(* IEC 61131-3 sources: ST2CPP/java/src/main/resources, 1 file *)

(* ---- iec_stdlib.st ---- *)
(* IEC 61131-3 标准类型转换函数声明 *)
(* 编译器生成 C++ 原型，运行时在 rt_plc.h 中实现 *)
(* 注意: TIME_OF_DAY/DATE_AND_TIME 类型暂不被 parser 识别，用 DINT/STRING 替代 *)

(* ─── 类型转换: X_TO_Y ─── *)
FUNCTION DINT_TO_TIME : TIME VAR_INPUT IN : DINT; END_VAR END_FUNCTION
FUNCTION UDINT_TO_DINT : DINT VAR_INPUT IN : UDINT; END_VAR END_FUNCTION
FUNCTION INT_TO_UDINT : UDINT VAR_INPUT IN : INT; END_VAR END_FUNCTION
FUNCTION UDINT_TO_TIME : TIME VAR_INPUT IN : UDINT; END_VAR END_FUNCTION
FUNCTION DINT_TO_UDINT : UDINT VAR_INPUT IN : DINT; END_VAR END_FUNCTION
FUNCTION TIME_TO_UDINT : UDINT VAR_INPUT IN : TIME; END_VAR END_FUNCTION
FUNCTION REAL_TO_DINT : DINT VAR_INPUT IN : REAL; END_VAR END_FUNCTION
FUNCTION REAL_TO_UDINT : UDINT VAR_INPUT IN : REAL; END_VAR END_FUNCTION
FUNCTION REAL_TO_DWORD : DWORD VAR_INPUT IN : REAL; END_VAR END_FUNCTION
FUNCTION REAL_TO_INT : INT VAR_INPUT IN : REAL; END_VAR END_FUNCTION
FUNCTION REAL_TO_WORD : WORD VAR_INPUT IN : REAL; END_VAR END_FUNCTION
FUNCTION REAL_TO_BYTE : BYTE VAR_INPUT IN : REAL; END_VAR END_FUNCTION
FUNCTION REAL_TO_TIME : TIME VAR_INPUT IN : REAL; END_VAR END_FUNCTION
FUNCTION REAL_TO_STRF : STRING VAR_INPUT IN : REAL; END_VAR END_FUNCTION
FUNCTION REAL_TO_STRING : STRING VAR_INPUT IN : REAL; END_VAR END_FUNCTION
FUNCTION INT_TO_DINT : DINT VAR_INPUT IN : INT; END_VAR END_FUNCTION
FUNCTION INT_TO_REAL : REAL VAR_INPUT IN : INT; END_VAR END_FUNCTION
FUNCTION INT_TO_DWORD : DWORD VAR_INPUT IN : INT; END_VAR END_FUNCTION
FUNCTION INT_TO_BYTE : BYTE VAR_INPUT IN : INT; END_VAR END_FUNCTION
FUNCTION INT_TO_WORD : WORD VAR_INPUT IN : INT; END_VAR END_FUNCTION
FUNCTION INT_TO_STRING : STRING VAR_INPUT IN : INT; END_VAR END_FUNCTION
FUNCTION INT_TO_TIME : TIME VAR_INPUT IN : INT; END_VAR END_FUNCTION
FUNCTION INT_TO_UINT : UINT VAR_INPUT IN : INT; END_VAR END_FUNCTION
FUNCTION DINT_TO_INT : INT VAR_INPUT IN : DINT; END_VAR END_FUNCTION
FUNCTION DINT_TO_REAL : REAL VAR_INPUT IN : DINT; END_VAR END_FUNCTION
FUNCTION DINT_TO_DWORD : DWORD VAR_INPUT IN : DINT; END_VAR END_FUNCTION
FUNCTION DINT_TO_WORD : WORD VAR_INPUT IN : DINT; END_VAR END_FUNCTION
FUNCTION DINT_TO_STRING : STRING VAR_INPUT IN : DINT; END_VAR END_FUNCTION
FUNCTION DWORD_TO_DINT : DINT VAR_INPUT IN : DWORD; END_VAR END_FUNCTION
FUNCTION DWORD_TO_INT : INT VAR_INPUT IN : DWORD; END_VAR END_FUNCTION
FUNCTION DWORD_TO_WORD : WORD VAR_INPUT IN : DWORD; END_VAR END_FUNCTION
FUNCTION DWORD_TO_BYTE : BYTE VAR_INPUT IN : DWORD; END_VAR END_FUNCTION
FUNCTION DWORD_TO_TIME : TIME VAR_INPUT IN : DWORD; END_VAR END_FUNCTION
FUNCTION DWORD_TO_UDINT : UDINT VAR_INPUT IN : DWORD; END_VAR END_FUNCTION
FUNCTION DWORD_TO_STRING : STRING VAR_INPUT IN : DWORD; END_VAR END_FUNCTION
FUNCTION DWORD_TO_STRB : STRING VAR_INPUT IN : DWORD; END_VAR END_FUNCTION
FUNCTION DWORD_TO_STRH : STRING VAR_INPUT IN : DWORD; END_VAR END_FUNCTION
FUNCTION DWORD_TO_STRF : STRING VAR_INPUT IN : DWORD; END_VAR END_FUNCTION
FUNCTION DW_TO_REAL : REAL VAR_INPUT IN : DWORD; END_VAR END_FUNCTION
FUNCTION UDINT_TO_REAL : REAL VAR_INPUT IN : UDINT; END_VAR END_FUNCTION
FUNCTION UDINT_TO_INT : INT VAR_INPUT IN : UDINT; END_VAR END_FUNCTION
FUNCTION UDINT_TO_DWORD : DWORD VAR_INPUT IN : UDINT; END_VAR END_FUNCTION
FUNCTION UDINT_TO_WORD : WORD VAR_INPUT IN : UDINT; END_VAR END_FUNCTION
FUNCTION UDINT_TO_BYTE : BYTE VAR_INPUT IN : UDINT; END_VAR END_FUNCTION
FUNCTION UDINT_TO_STRING : STRING VAR_INPUT IN : UDINT; END_VAR END_FUNCTION
FUNCTION UDINT_TO_UINT : UINT VAR_INPUT IN : UDINT; END_VAR END_FUNCTION
FUNCTION WORD_TO_DINT : DINT VAR_INPUT IN : WORD; END_VAR END_FUNCTION
FUNCTION WORD_TO_INT : INT VAR_INPUT IN : WORD; END_VAR END_FUNCTION
FUNCTION WORD_TO_DWORD : DWORD VAR_INPUT IN : WORD; END_VAR END_FUNCTION
FUNCTION WORD_TO_BYTE : BYTE VAR_INPUT IN : WORD; END_VAR END_FUNCTION
FUNCTION WORD_TO_UDINT : UDINT VAR_INPUT IN : WORD; END_VAR END_FUNCTION
FUNCTION WORD_TO_UINT : UINT VAR_INPUT IN : WORD; END_VAR END_FUNCTION
FUNCTION WORD_TO_STRING : STRING VAR_INPUT IN : WORD; END_VAR END_FUNCTION
FUNCTION BYTE_TO_DINT : DINT VAR_INPUT IN : BYTE; END_VAR END_FUNCTION
FUNCTION BYTE_TO_INT : INT VAR_INPUT IN : BYTE; END_VAR END_FUNCTION
FUNCTION BYTE_TO_DWORD : DWORD VAR_INPUT IN : BYTE; END_VAR END_FUNCTION
FUNCTION BYTE_TO_WORD : WORD VAR_INPUT IN : BYTE; END_VAR END_FUNCTION
FUNCTION BYTE_TO_UDINT : UDINT VAR_INPUT IN : BYTE; END_VAR END_FUNCTION
FUNCTION BYTE_TO_UINT : UINT VAR_INPUT IN : BYTE; END_VAR END_FUNCTION
FUNCTION BYTE_TO_USINT : USINT VAR_INPUT IN : BYTE; END_VAR END_FUNCTION
FUNCTION BYTE_TO_STRING : STRING VAR_INPUT IN : BYTE; END_VAR END_FUNCTION
FUNCTION BYTE_TO_STRB : STRING VAR_INPUT IN : BYTE; END_VAR END_FUNCTION
FUNCTION BYTE_TO_STRH : STRING VAR_INPUT IN : BYTE; END_VAR END_FUNCTION
FUNCTION BYTE_TO_BITS : STRING VAR_INPUT IN : BYTE; END_VAR END_FUNCTION
FUNCTION BYTE_TO_GRAY : BYTE VAR_INPUT IN : BYTE; END_VAR END_FUNCTION
FUNCTION BYTE_TO_TIME2 : TIME VAR_INPUT IN : BYTE; END_VAR END_FUNCTION
FUNCTION UINT_TO_DINT : DINT VAR_INPUT IN : UINT; END_VAR END_FUNCTION
FUNCTION UINT_TO_INT : INT VAR_INPUT IN : UINT; END_VAR END_FUNCTION
FUNCTION UINT_TO_DWORD : DWORD VAR_INPUT IN : UINT; END_VAR END_FUNCTION
FUNCTION UINT_TO_BYTE : BYTE VAR_INPUT IN : UINT; END_VAR END_FUNCTION
FUNCTION UINT_TO_WORD : WORD VAR_INPUT IN : UINT; END_VAR END_FUNCTION
FUNCTION UINT_TO_UDINT : UDINT VAR_INPUT IN : UINT; END_VAR END_FUNCTION
FUNCTION UINT_TO_REAL : REAL VAR_INPUT IN : UINT; END_VAR END_FUNCTION
FUNCTION USINT_TO_INT : INT VAR_INPUT IN : USINT; END_VAR END_FUNCTION
FUNCTION USINT_TO_BYTE : BYTE VAR_INPUT IN : USINT; END_VAR END_FUNCTION
FUNCTION USINT_TO_REAL : REAL VAR_INPUT IN : USINT; END_VAR END_FUNCTION
FUNCTION USINT_TO_DINT : DINT VAR_INPUT IN : USINT; END_VAR END_FUNCTION
FUNCTION SINT_TO_INT : INT VAR_INPUT IN : SINT; END_VAR END_FUNCTION
FUNCTION SINT_TO_DINT : DINT VAR_INPUT IN : SINT; END_VAR END_FUNCTION
FUNCTION STRING_TO_TIME : TIME VAR_INPUT IN : STRING; END_VAR END_FUNCTION
FUNCTION STRING_TO_INT : INT VAR_INPUT IN : STRING; END_VAR END_FUNCTION
FUNCTION STRING_TO_REAL : REAL VAR_INPUT IN : STRING; END_VAR END_FUNCTION
FUNCTION STRING_TO_DWORD : DWORD VAR_INPUT IN : STRING; END_VAR END_FUNCTION
FUNCTION STRING_TO_WORD : WORD VAR_INPUT IN : STRING; END_VAR END_FUNCTION
FUNCTION STRING_TO_UDINT : UDINT VAR_INPUT IN : STRING; END_VAR END_FUNCTION
FUNCTION STRING_TO_URL : STRING VAR_INPUT IN : STRING; END_VAR END_FUNCTION
FUNCTION STRING_TO_BUFFER : STRING VAR_INPUT IN : STRING; END_VAR END_FUNCTION
FUNCTION BOOL_TO_BYTE : BYTE VAR_INPUT IN : BOOL; END_VAR END_FUNCTION
FUNCTION BOOL_TO_INT : INT VAR_INPUT IN : BOOL; END_VAR END_FUNCTION
FUNCTION BOOL_TO_DWORD : DWORD VAR_INPUT IN : BOOL; END_VAR END_FUNCTION
FUNCTION BOOL_TO_UDINT : UDINT VAR_INPUT IN : BOOL; END_VAR END_FUNCTION
FUNCTION BOOL_TO_STRING : STRING VAR_INPUT IN : BOOL; END_VAR END_FUNCTION
FUNCTION TIME_TO_DINT : DINT VAR_INPUT IN : TIME; END_VAR END_FUNCTION
FUNCTION TIME_TO_INT : INT VAR_INPUT IN : TIME; END_VAR END_FUNCTION
FUNCTION TIME_TO_DWORD : DWORD VAR_INPUT IN : TIME; END_VAR END_FUNCTION
FUNCTION TIME_TO_REAL : REAL VAR_INPUT IN : TIME; END_VAR END_FUNCTION
FUNCTION TIME_TO_TOD : STRING VAR_INPUT IN : TIME; END_VAR END_FUNCTION
FUNCTION TOD_TO_TIME : TIME VAR_INPUT IN : STRING; END_VAR END_FUNCTION
FUNCTION TOD_TO_REAL2 : REAL VAR_INPUT IN : STRING; END_VAR END_FUNCTION
FUNCTION DATE_TO_UDINT : UDINT VAR_INPUT IN : INT; END_VAR END_FUNCTION
FUNCTION DATE_TO_DT : INT VAR_INPUT IN : INT; END_VAR END_FUNCTION
FUNCTION DATE_TO_STRING2 : STRING VAR_INPUT IN : INT; END_VAR END_FUNCTION
FUNCTION DATE_TO_REAL2 : REAL VAR_INPUT IN : INT; END_VAR END_FUNCTION
FUNCTION DATE_TO_DWORD2 : DWORD VAR_INPUT IN : INT; END_VAR END_FUNCTION
FUNCTION DT_TO_DATE : INT VAR_INPUT IN : INT; END_VAR END_FUNCTION
FUNCTION DT_TO_DATE2 : INT VAR_INPUT IN : INT; END_VAR END_FUNCTION
FUNCTION DT_TO_TOD2 : STRING VAR_INPUT IN : INT; END_VAR END_FUNCTION
FUNCTION DT_TO_SDT : INT VAR_INPUT IN : INT; END_VAR END_FUNCTION
FUNCTION DT_TO_STRF : STRING VAR_INPUT IN : INT; END_VAR END_FUNCTION
FUNCTION SDT_TO_DATE : INT VAR_INPUT IN : INT; END_VAR END_FUNCTION
FUNCTION SDT_TO_DT : INT VAR_INPUT IN : INT; END_VAR END_FUNCTION
FUNCTION SDT_TO_TOD : STRING VAR_INPUT IN : INT; END_VAR END_FUNCTION

(* ─── 字符串操作 ─── *)
FUNCTION CONCAT : STRING VAR_INPUT A : STRING; B : STRING; END_VAR END_FUNCTION
FUNCTION LEN : DINT VAR_INPUT S : STRING; END_VAR END_FUNCTION
FUNCTION LEFT : STRING VAR_INPUT S : STRING; L : DINT; END_VAR END_FUNCTION
FUNCTION RIGHT : STRING VAR_INPUT S : STRING; L : DINT; END_VAR END_FUNCTION
FUNCTION MID : STRING VAR_INPUT S : STRING; L : DINT; P : DINT; END_VAR END_FUNCTION
FUNCTION INSERT : STRING VAR_INPUT S : STRING; INS : STRING; P : DINT; END_VAR END_FUNCTION
FUNCTION DELETE : STRING VAR_INPUT S : STRING; L : DINT; P : DINT; END_VAR END_FUNCTION
FUNCTION REPLACE : STRING VAR_INPUT S : STRING; L : DINT; P : DINT; R : STRING; END_VAR END_FUNCTION
FUNCTION FIND : DINT VAR_INPUT S : STRING; SUBSTR : STRING; END_VAR END_FUNCTION
FUNCTION STR_EQ : BOOL VAR_INPUT A : STRING; B : STRING; END_VAR END_FUNCTION
FUNCTION STR_NE : BOOL VAR_INPUT A : STRING; B : STRING; END_VAR END_FUNCTION
FUNCTION STR_LT : BOOL VAR_INPUT A : STRING; B : STRING; END_VAR END_FUNCTION
FUNCTION STR_LE : BOOL VAR_INPUT A : STRING; B : STRING; END_VAR END_FUNCTION
FUNCTION STR_GT : BOOL VAR_INPUT A : STRING; B : STRING; END_VAR END_FUNCTION
FUNCTION STR_GE : BOOL VAR_INPUT A : STRING; B : STRING; END_VAR END_FUNCTION

(* ─── 数学函数 ─── *)
FUNCTION ABS : REAL VAR_INPUT X : REAL; END_VAR END_FUNCTION
FUNCTION SQRT : REAL VAR_INPUT X : REAL; END_VAR END_FUNCTION
FUNCTION LN : REAL VAR_INPUT X : REAL; END_VAR END_FUNCTION
FUNCTION LOG : REAL VAR_INPUT X : REAL; END_VAR END_FUNCTION
FUNCTION EXP : REAL VAR_INPUT X : REAL; END_VAR END_FUNCTION
FUNCTION EXPT : REAL VAR_INPUT X : REAL; Y : REAL; END_VAR END_FUNCTION
FUNCTION SIN : REAL VAR_INPUT X : REAL; END_VAR END_FUNCTION
FUNCTION COS : REAL VAR_INPUT X : REAL; END_VAR END_FUNCTION
FUNCTION TAN : REAL VAR_INPUT X : REAL; END_VAR END_FUNCTION
FUNCTION ASIN : REAL VAR_INPUT X : REAL; END_VAR END_FUNCTION
FUNCTION ACOS : REAL VAR_INPUT X : REAL; END_VAR END_FUNCTION
FUNCTION ATAN : REAL VAR_INPUT X : REAL; END_VAR END_FUNCTION
FUNCTION ATAN2 : REAL VAR_INPUT Y : REAL; X : REAL; END_VAR END_FUNCTION

(* ─── 标准功能块 ─── *)
FUNCTION_BLOCK SR
    VAR_INPUT S1 : BOOL; R : BOOL; END_VAR
    VAR_OUTPUT Q1 : BOOL; END_VAR
END_FUNCTION_BLOCK

FUNCTION_BLOCK RS
    VAR_INPUT S : BOOL; R1 : BOOL; END_VAR
    VAR_OUTPUT Q1 : BOOL; END_VAR
END_FUNCTION_BLOCK

FUNCTION_BLOCK R_TRIG
    VAR_INPUT CLK : BOOL; END_VAR
    VAR_OUTPUT Q : BOOL; END_VAR
    VAR lastCLK : BOOL; END_VAR
END_FUNCTION_BLOCK

FUNCTION_BLOCK F_TRIG
    VAR_INPUT CLK : BOOL; END_VAR
    VAR_OUTPUT Q : BOOL; END_VAR
    VAR lastCLK : BOOL; END_VAR
END_FUNCTION_BLOCK

FUNCTION_BLOCK CTU
    VAR_INPUT CU : BOOL; R : BOOL; PV : INT; END_VAR
    VAR_OUTPUT Q : BOOL; CV : INT; END_VAR
    VAR lastCU : BOOL; END_VAR
END_FUNCTION_BLOCK

FUNCTION_BLOCK CTD
    VAR_INPUT CD : BOOL; LD : BOOL; PV : INT; END_VAR
    VAR_OUTPUT Q : BOOL; CV : INT; END_VAR
    VAR lastCD : BOOL; END_VAR
END_FUNCTION_BLOCK

FUNCTION_BLOCK CTUD
    VAR_INPUT CU : BOOL; CD : BOOL; R : BOOL; LD : BOOL; PV : INT; END_VAR
    VAR_OUTPUT QU : BOOL; QD : BOOL; CV : INT; END_VAR
    VAR lastCU : BOOL; lastCD : BOOL; END_VAR
END_FUNCTION_BLOCK

FUNCTION_BLOCK TP
    VAR_INPUT IN : BOOL; PT : TIME; END_VAR
    VAR_OUTPUT Q : BOOL; ET : TIME; END_VAR
    VAR lastInput : BOOL; END_VAR
END_FUNCTION_BLOCK

FUNCTION_BLOCK TON
    VAR_INPUT IN : BOOL; PT : TIME; END_VAR
    VAR_OUTPUT Q : BOOL; ET : TIME; END_VAR
END_FUNCTION_BLOCK

FUNCTION_BLOCK TOF
    VAR_INPUT IN : BOOL; PT : TIME; END_VAR
    VAR_OUTPUT Q : BOOL; ET : TIME; END_VAR
END_FUNCTION_BLOCK

(* ─── 选择函数 ─── *)
FUNCTION SEL : REAL VAR_INPUT G : BOOL; IN0 : REAL; IN1 : REAL; END_VAR END_FUNCTION
FUNCTION MUX : REAL VAR_INPUT K : INT; IN0 : REAL; IN1 : REAL; IN2 : REAL; IN3 : REAL; END_VAR END_FUNCTION
FUNCTION LIMIT : REAL VAR_INPUT MN : REAL; IN : REAL; MX : REAL; END_VAR END_FUNCTION
FUNCTION MAX : REAL VAR_INPUT IN0 : REAL; IN1 : REAL; END_VAR END_FUNCTION
FUNCTION MIN : REAL VAR_INPUT IN0 : REAL; IN1 : REAL; END_VAR END_FUNCTION
(* ─── 位操作 ─── *)
FUNCTION SHL : DWORD VAR_INPUT IN : DWORD; N : INT; END_VAR END_FUNCTION
FUNCTION SHR : DWORD VAR_INPUT IN : DWORD; N : INT; END_VAR END_FUNCTION
FUNCTION ROL : DWORD VAR_INPUT IN : DWORD; N : INT; END_VAR END_FUNCTION
FUNCTION ROR : DWORD VAR_INPUT IN : DWORD; N : INT; END_VAR END_FUNCTION

(* ─── 其他 ─── *)
FUNCTION MOVE : REAL VAR_INPUT IN : REAL; END_VAR END_FUNCTION
FUNCTION TRUNC : REAL VAR_INPUT IN : REAL; END_VAR END_FUNCTION
FUNCTION BCD_TO_INT : INT VAR_INPUT IN : BYTE; END_VAR END_FUNCTION
FUNCTION INT_TO_BCD : BYTE VAR_INPUT IN : INT; END_VAR END_FUNCTION
FUNCTION GRAY_TO_BYTE : BYTE VAR_INPUT IN : BYTE; END_VAR END_FUNCTION
FUNCTION FLOOR : INT VAR_INPUT X : REAL; END_VAR END_FUNCTION
